TYPE ExampleCylinderConfig : 
STRUCT
    TimeToReachHomePosition : TIME := T#10S;
    TimeToReachWorkPosition : TIME := T#10S;
END_STRUCT
END_TYPE

(* stored: Version 1.1.0.1, ProductVersion 3.1.4024.9
   DUT ExampleCylinderConfig: Id {50189353-104d-0512-3a89-7ec2456d96b9} *)
